FUNCTION INTERNAL Tc2MC2_TO_Tco_SetPositionMode : BOOL
VAR_INPUT
    Tc2MC2SetPositionMode : BOOL;
END_VAR
VAR_IN_OUT
    TcoSetPositionMode : eSetPositionMode;
END_VAR

IF Tc2MC2SetPositionMode THEN
    TcoSetPositionMode := eSetPositionMode.Absolute;
    Tc2MC2_TO_Tco_SetPositionMode := TRUE;
ELSE
    TcoSetPositionMode := eSetPositionMode.Relative;
    Tc2MC2_TO_Tco_SetPositionMode := TRUE;
END_IF

END_FUNCTION

(* stored: Version 1.1.0.1, ProductVersion 3.1.4024.6
   POU Tc2MC2_TO_Tco_SetPositionMode: Id {2b9e2350-25a2-0951-3eb1-e32c7b27e4e1}, SpecialFunc None *)
